(*
A broadcastable wrapper for a `REAL` value. 
*)
INTERFACE I_RealArg EXTENDS I_Arg

(*
Reads the internal value.
*)
PROPERTY Get : REAL
GET
END_GET
END_PROPERTY

(*
Returns TRUE if the value is mutable.
*)
PROPERTY IsMut : BOOL
GET
END_GET
END_PROPERTY

(*
Modifies the internal value.  
Returns:
- `Ok` - Upon successful modification.
- `Error` - If mutability is disabled.
*)
METHOD Set : Result
VAR_INPUT
	newVal		: REAL;
END_VAR
END_METHOD

END_INTERFACE

(* stored: Version 1.1.0.1
   Itf I_RealArg: Id {60c82db8-698f-4c6d-b0fd-941beb5230f0}
   Property Get: Id {91293321-100d-499c-8411-2b0ee19089cc}
   Get Get: Id {7a833035-9daa-4a56-8ec8-904e616a366f}
   Property IsMut: Id {b66fe8de-1804-4144-81cb-a2cc027c6929}
   Get Get: Id {decb652a-d8d7-4379-9f8b-30244e3eff36}
   Method Set: Id {0417b581-50d8-4642-bf41-95b4f3b1598f} *)
